TYPE ST_Beckhoff_Drive_AX8206 :
STRUCT
	
	// Process
	T_RESET : F_TRIG ;
	
	// Drive <=> PLC		
	AxisRef : AXIS_REF;
		
END_STRUCT
END_TYPE

(* stored: Version 1.1.0.1, ProductVersion 3.1.4024.13
   DUT ST_Beckhoff_Drive_AX8206: Id {92a89cf8-edf0-41a1-a6cf-524fe68e289b} *)
